FUNCTION_BLOCK L0_StateHandler (* Basic Function Block Type *)
  (* Standard: 61499-2; Description: FB to handle CNC state changes *)
  (* Version 0.0, 2014-09-01, EQUEROL, UJI *)
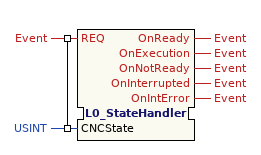
  EVENT_INPUT
    REQ WITH CNCState; (* Normal Execution Request *)
  END_EVENT
  EVENT_OUTPUT
    OnReady; (* Event Output when CNC is ready *)
    OnExecution; (* Event Output when CNC is executing *)
    OnNotReady; (* Event Output when CNC is Not Ready *)
    OnInterrupted; (* Event Output when CNC is interrupted *)
    OnIntError; (* Event Output when CNC is interrupted by error *)
  END_EVENT
  VAR_INPUT
    CNCState : USINT; (* CNC State *)
  END_VAR
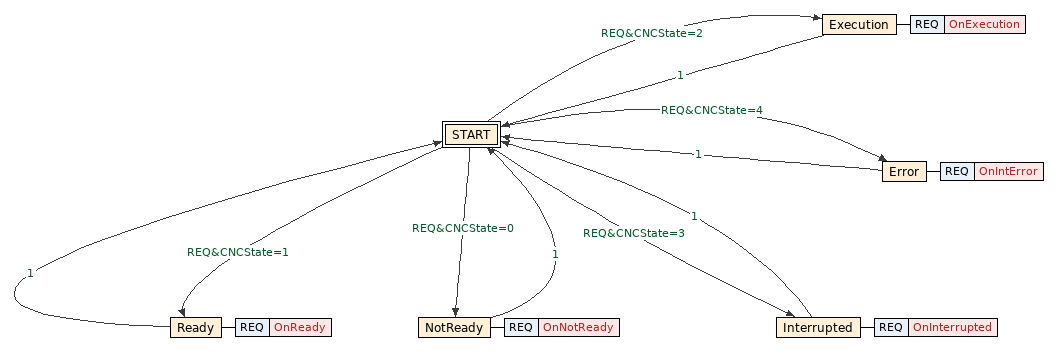
  EC_STATES
    START; (* Initial State *)
    Ready : REQ -> OnReady; (* Normal execution *)
    NotReady : REQ -> OnNotReady;
    Interrupted : REQ -> OnInterrupted;
    Error : REQ -> OnIntError;
    Execution : REQ -> OnExecution;
  END_STATES
  EC_TRANSITIONS
    START TO Ready := REQ&CNCState=1;
    Ready TO START := 1;
    START TO NotReady := REQ&CNCState=0;
    NotReady TO START := 1;
    START TO Interrupted := REQ&CNCState=3;
    Interrupted TO START := 1;
    START TO Error := REQ&CNCState=4;
    Error TO START := 1;
    Execution TO START := 1;
    START TO Execution := REQ&CNCState=2;
  END_TRANSITIONS
  ALGORITHM REQ IN ST: (* Normally executed algorithm *)

  END_ALGORITHM
END_FUNCTION_BLOCK
